TYPE TEST :
UNION
	arrByte 		:ARRAY[0..15] OF BYTE;
	arrWord			:WORD ; 
END_UNION
END_TYPE

(* stored: Version 1.1.0.1
   DUT TEST: Id {98b73179-2ce5-4a59-844f-3ad4760502f2} *)
